{attribute 'qualified_only'}
{attribute 'strict'}
TYPE E_Conveyor :
(
	enum_member := 0
);
END_TYPE

(* stored: Version 1.1.0.1, ProductVersion 3.1.4024.12
   DUT E_Conveyor: Id {663bde4a-a10e-4dba-ba45-b90e8e5263b8} *)
